INTERFACE I_ImageBlender

METHOD Mix
VAR_INPUT
	ImageBottomLayer : ITcVnImage;
	ImageTopLayer	 : ITcVnImage;
END_VAR
END_METHOD

END_INTERFACE

(* stored: Version 1.1.0.1
   Itf I_ImageBlender: Id {8eb2b565-bbbe-4fa3-b1c3-abe920cba2eb}
   Method Mix: Id {0784042c-e250-42ed-b9f4-2ea76e60a256} *)
